FUNCTION "oRMain" : Void
{ S7_Optimized_Access := 'TRUE' }
VERSION : 0.8
   VAR_TEMP
      index : "tIndex";
      location : Int;
      i : Int;
   END_VAR


BEGIN
	"fSizeArray"(size => #index.qty,
	             io_Array := "dbArchiveEquipRectifier".equipmentRectifier);
	#location := 1200;

	//Call all equipment
	FOR #index.acc := 1 TO #index.qty DO
	    "fRectifier"(index := #index,
	                location := #location);
	END_FOR;
END_FUNCTION

